// TIA Portal V18 export
// export: Created 2026-01-09T11:31:53.6972974Z, ExportSetting WithDefaults, DisplayName Totally Integrated Automation Portal, DisplayVersion V18 Update 5, DisplayName TIA Portal Openness, DisplayVersion V18 Update 5, DisplayName TIA Portal Teamcenter Gateway, DisplayVersion V18, DisplayName TIA Portal Version Control Interface, DisplayVersion V18, DisplayName SINAMICS Startdrive Advanced, DisplayVersion V18 SP2 Update 1, DisplayName SINAMICS Startdrive G110M, G120, G120C, G120D, G120P, G115D, DisplayVersion V18 SP2 Update 1, DisplayName SINAMICS Startdrive G130, G150, S120, S150, SINAMICS MV, S210, G220, S200, DisplayVersion V18 SP2 Update 1, DisplayName STEP 7 Professional, DisplayVersion V18 Update 5, DisplayName STEP 7 Safety, DisplayVersion V18, DisplayName WinCC Professional, DisplayVersion V18 Update 5
TagTable "ST350_PartData"
  PartData_Interface_DB_PartDataID : Int  (PLC tag PartData_Interface_DB.PartDataID, CPU S71500-2PN_TP700, 1 s)
  PartData_Interface_DB_PartData{1}_PartDataHMI : PartDataHMI  (PLC tag PartData_Interface_DB.PartData[1].PartDataHMI, CPU S71500-2PN_TP700, 1 s)
    TagStructureMember "PartQuality"
    TagStructureMember "BoxDisplayID"
    TagStructureMember "PartQualitySet"
    TagStructureMember "CMD"
      TagStructureMember "ClearCurrentBox"
      TagStructureMember "ClearAllBox"
      TagStructureMember "PartQuality+1"
      TagStructureMember "PartQuality-1"
      TagStructureMember "PartQualityAck"
    TagStructureMember "Waring"
      TagStructureMember "Insufficient"
      TagStructureMember "BufferBoxFull"
      TagStructureMember "ScannCodeInvalid"
    TagStructureMember "PartDataDispaly"
      TagStructureMember "PartCode"
      TagStructureMember "PartCode_Len"
      TagStructureMember "SupplierID"
      TagStructureMember "MaterialType"
      TagStructureMember "PO_ID"
      TagStructureMember "BatchID"
      TagStructureMember "Quality"
      TagStructureMember "Cartons"
      TagStructureMember "PartQuality"
  PartData_Interface_DB_PartData{2}_PartDataHMI : PartDataHMI  (PLC tag PartData_Interface_DB.PartData[2].PartDataHMI, CPU S71500-2PN_TP700, 1 s)
    TagStructureMember "PartQuality"
    TagStructureMember "BoxDisplayID"
    TagStructureMember "PartQualitySet"
    TagStructureMember "CMD"
      TagStructureMember "ClearCurrentBox"
      TagStructureMember "ClearAllBox"
      TagStructureMember "PartQuality+1"
      TagStructureMember "PartQuality-1"
      TagStructureMember "PartQualityAck"
    TagStructureMember "Waring"
      TagStructureMember "Insufficient"
      TagStructureMember "BufferBoxFull"
      TagStructureMember "ScannCodeInvalid"
    TagStructureMember "PartDataDispaly"
      TagStructureMember "PartCode"
      TagStructureMember "PartCode_Len"
      TagStructureMember "SupplierID"
      TagStructureMember "MaterialType"
      TagStructureMember "PO_ID"
      TagStructureMember "BatchID"
      TagStructureMember "Quality"
      TagStructureMember "Cartons"
      TagStructureMember "PartQuality"
  PartData_Interface_DB_PartCMD{1}_Set(1) : Bool  (PLC tag PartData_Interface_DB.PartCMD[1].Set, CPU S71500-2PN_TP700, 1 s)
  PartData_Interface_DB_PartCMD{1}_Use(1) : Bool  (PLC tag PartData_Interface_DB.PartCMD[1].Use, CPU S71500-2PN_TP700, 1 s)
  PartData_Interface_DB_PartCMD{2}_Set : Bool  (PLC tag PartData_Interface_DB.PartCMD[2].Set, CPU S71500-2PN_TP700, 1 s)
  PartData_Interface_DB_PartCMD{2}_Use : Bool  (PLC tag PartData_Interface_DB.PartCMD[2].Use, CPU S71500-2PN_TP700, 1 s)
